{attribute addProperty BoxType "KL3208-0002"}
{attribute addProperty Id "Channel_1Channel_B0A8062F00Channel_2Channel_B0A8062F00Channel_3Channel_B0A8062F00Channel_4Channel_B0A8062F00"}
{attribute addProperty CRC "2945616803"}
{attribute addProperty SizeInBites "0"}
{attribute addProperty SizeInBytes "0"}
TYPE KL_AF928BA3 :
STRUCT
	{attribute addProperty Name "Channel_1"}
	Channel_1 : Channel_B0A8062F;
	{attribute addProperty Name "Channel_2"}
	Channel_2 : Channel_B0A8062F;
	{attribute addProperty Name "Channel_3"}
	Channel_3 : Channel_B0A8062F;
	{attribute addProperty Name "Channel_4"}
	Channel_4 : Channel_B0A8062F;
END_STRUCT
END_TYPE

(* stored: Version 1.2.0.0, ProductVersion 3.1.4024.9
   DUT KL_AF928BA3: Id {e3280aa3-0922-4215-9274-a1da4128be57} *)
